VISUALIZATION Settings_PNG  // 800x480
END_VISUALIZATION

(* stored: Version 1.1.0.1, ProductVersion 3.1.4024.5
   Visu Settings_PNG: Id {902dec27-9ce0-460e-9363-33508825ca96} *)
